FUNCTION F_HMI_BUSY_TO_COLOR : T_HMI_COLORS
VAR_IN_OUT
    fbBusyStatus : FB_HMI_BUSY_STATUS;
END_VAR
VAR_OUTPUT
END_VAR
VAR
END_VAR

IF fbBusyStatus.bIdle THEN
    F_HMI_BUSY_TO_COLOR.fg := E_HMI_COLORS.BLACK;
    F_HMI_BUSY_TO_COLOR.bg := E_HMI_COLORS.GREEN;
ELSIF fbBusyStatus.bBusy THEN
	F_HMI_BUSY_TO_COLOR.fg := E_HMI_COLORS.WHITE;
	F_HMI_BUSY_TO_COLOR.bg := E_HMI_COLORS.BLUE;
ELSE
	F_HMI_BUSY_TO_COLOR.fg := E_HMI_COLORS.BLACK;
	F_HMI_BUSY_TO_COLOR.bg := E_HMI_COLORS.GRAY;
END_IF

END_FUNCTION

(* stored: Version 1.1.0.1, ProductVersion 3.1.4024.14
   POU F_HMI_BUSY_TO_COLOR: Id {a66562d8-d268-4b3f-a05d-c93ec2e0b4c2}, SpecialFunc None *)
